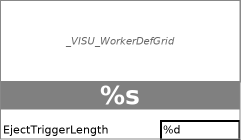
VISUALIZATION _VISU_WorkerDefGrid_Verify  // 241x140
VAR_IN_OUT
		m_Inst : FB_WorkerDefGrid_Verify;
END_VAR
    Frame (0,0 241x82)
        shows _VISU_WorkerDefGrid(m_Inst := m_Inst)
    Rectangle (0,80 240x30), "%s", text variable: m_Inst._name, colour toggle: m_Inst._pAttachedCt <> 0
    Rectangle (0,120 160x20), "EjectTriggerLength"
    Rectangle (160,120 80x20), "%d", text variable: m_Inst.tpEjectPulse.PT
        OnMouseDown: write the text variable via Default
END_VISUALIZATION

(* stored: Version 1.1.0.1, ProductVersion 3.1.4024.11
   Visu _VISU_WorkerDefGrid_Verify: Id {c49ee8c0-c797-4c5e-a870-e0f74b5ccead} *)
